Fanuc KAREL source: port_AIN.kl

PROGRAM TP
%NOLOCKGROUP
VAR
 x: INTEGER
BEGIN
 x = AIN[3]
END TP
